FUNCTION_BLOCK I_Lighting (* Lighting Data LD *)
  (* Standard: ISO 11783-7; Classification: PGN 65088; Function: Lighting Data LD; Description: Copyright (c) 2024 HR Agrartechnik GmbH This program and the accompanying materials are made available under the terms of the Eclipse Public License 2.0 which is available at https://www.eclipse.org/legal/epl-2.0/ SPDX-License-Identifier: EPL-2.0 Message providing the status of all lighting functions of a tractor and connected implements. https://docs.ms-muc-docs.de/projects/isobus-other-docs/de/latest/PGN/PGN_65088.html *)
  (* Version 1.0, 2024-07-09, Franz Höpfinger, HR Agrartechnik GmbH *)
  PACKAGE isobus::tecu;
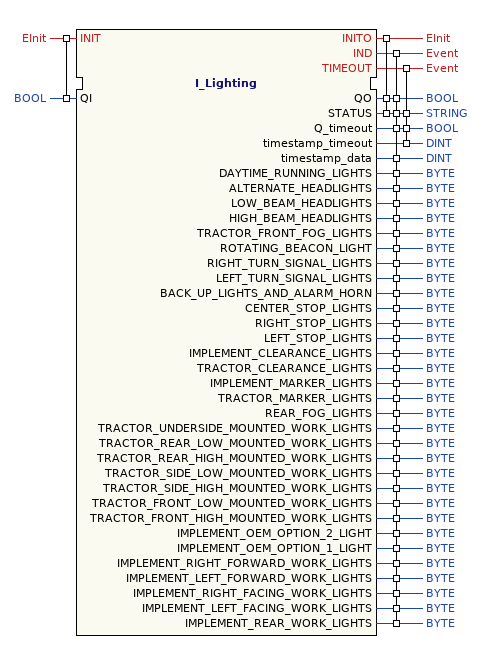
  EVENT_INPUT
    INIT : EInit WITH QI; (* Service Initialization *)
  END_EVENT
  EVENT_OUTPUT
    INITO : EInit WITH QO, STATUS; (* Initialization Confirm *)
    IND WITH QO, timestamp_data, STATUS, Q_timeout, DAYTIME_RUNNING_LIGHTS, ALTERNATE_HEADLIGHTS, LOW_BEAM_HEADLIGHTS, HIGH_BEAM_HEADLIGHTS, TRACTOR_FRONT_FOG_LIGHTS, ROTATING_BEACON_LIGHT, RIGHT_TURN_SIGNAL_LIGHTS, LEFT_TURN_SIGNAL_LIGHTS, BACK_UP_LIGHTS_AND_ALARM_HORN, CENTER_STOP_LIGHTS, RIGHT_STOP_LIGHTS, LEFT_STOP_LIGHTS, IMPLEMENT_CLEARANCE_LIGHTS, TRACTOR_CLEARANCE_LIGHTS, IMPLEMENT_MARKER_LIGHTS, TRACTOR_MARKER_LIGHTS, REAR_FOG_LIGHTS, TRACTOR_UNDERSIDE_MOUNTED_WORK_LIGHTS, TRACTOR_REAR_LOW_MOUNTED_WORK_LIGHTS, TRACTOR_REAR_HIGH_MOUNTED_WORK_LIGHTS, TRACTOR_SIDE_LOW_MOUNTED_WORK_LIGHTS, TRACTOR_SIDE_HIGH_MOUNTED_WORK_LIGHTS, TRACTOR_FRONT_LOW_MOUNTED_WORK_LIGHTS, TRACTOR_FRONT_HIGH_MOUNTED_WORK_LIGHTS, IMPLEMENT_OEM_OPTION_2_LIGHT, IMPLEMENT_OEM_OPTION_1_LIGHT, IMPLEMENT_RIGHT_FORWARD_WORK_LIGHTS, IMPLEMENT_LEFT_FORWARD_WORK_LIGHTS, IMPLEMENT_RIGHT_FACING_WORK_LIGHTS, IMPLEMENT_LEFT_FACING_WORK_LIGHTS, IMPLEMENT_REAR_WORK_LIGHTS; (* Indication from Resource *)
    TIMEOUT WITH timestamp_timeout, STATUS, Q_timeout;
  END_EVENT
  VAR_INPUT
    QI : BOOL; (* Event Input Qualifier *)
  END_VAR
  VAR_OUTPUT
    QO : BOOL; (* Event Output Qualifier *)
    STATUS : STRING;
    Q_timeout : BOOL;
    timestamp_timeout : DINT;
    timestamp_data : DINT;
    DAYTIME_RUNNING_LIGHTS : BYTE := BYTE#16#FF; (* Daytime running lights 2-bit QUARTER value (see Attributes for Details) *) {SET_ATTRIBUTE(SPN, 2404)} {SET_ATTRIBUTE(SP_Name, 'Daytime running lights')} {SET_ATTRIBUTE(SP_Position_In_PG, '1.1')} {SET_ATTRIBUTE(SP_Length, 2)} (* 2 bits *) {SET_ATTRIBUTE(Scaling, '4 states/2 bit')} {SET_ATTRIBUTE(Offset, )} {SET_ATTRIBUTE(Link, 'https://docs.ms-muc-docs.de/projects/isobus-other-docs/de/latest/PGN/PGN_65088.html#spn-2404-daytime-running-lights')}
    ALTERNATE_HEADLIGHTS : BYTE := BYTE#16#FF; (* Alternate headlights 2-bit QUARTER value (see Attributes for Details) *) {SET_ATTRIBUTE(SPN, 2352)} {SET_ATTRIBUTE(SP_Name, 'Alternate headlights')} {SET_ATTRIBUTE(SP_Position_In_PG, '1.3')} {SET_ATTRIBUTE(SP_Length, 2)} (* 2 bits *) {SET_ATTRIBUTE(Scaling, '4 states/2 bit')} {SET_ATTRIBUTE(Offset, )} {SET_ATTRIBUTE(Link, 'https://docs.ms-muc-docs.de/projects/isobus-other-docs/de/latest/PGN/PGN_65088.html#spn-2352-alternate-headlights')}
    LOW_BEAM_HEADLIGHTS : BYTE := BYTE#16#FF; (* Low-beam headlights 2-bit QUARTER value (see Attributes for Details) *) {SET_ATTRIBUTE(SPN, 2350)} {SET_ATTRIBUTE(SP_Name, 'Low-beam headlights')} {SET_ATTRIBUTE(SP_Position_In_PG, '1.5')} {SET_ATTRIBUTE(SP_Length, 2)} (* 2 bits *) {SET_ATTRIBUTE(Scaling, '4 states/2 bit')} {SET_ATTRIBUTE(Offset, )} {SET_ATTRIBUTE(Link, 'https://docs.ms-muc-docs.de/projects/isobus-other-docs/de/latest/PGN/PGN_65088.html#spn-2350-low-beam-headlights')}
    HIGH_BEAM_HEADLIGHTS : BYTE := BYTE#16#FF; (* High-beam headlights 2-bit QUARTER value (see Attributes for Details) *) {SET_ATTRIBUTE(SPN, 2348)} {SET_ATTRIBUTE(SP_Name, 'High-beam headlights')} {SET_ATTRIBUTE(SP_Position_In_PG, '1.7')} {SET_ATTRIBUTE(SP_Length, 2)} (* 2 bits *) {SET_ATTRIBUTE(Scaling, '4 states/2 bit')} {SET_ATTRIBUTE(Offset, )} {SET_ATTRIBUTE(Link, 'https://docs.ms-muc-docs.de/projects/isobus-other-docs/de/latest/PGN/PGN_65088.html#spn-2348-high-beam-headlights')}
    TRACTOR_FRONT_FOG_LIGHTS : BYTE := BYTE#16#FF; (* Tractor front fog lights 2-bit QUARTER value (see Attributes for Details) *) {SET_ATTRIBUTE(SPN, 2388)} {SET_ATTRIBUTE(SP_Name, 'Tractor front fog lights')} {SET_ATTRIBUTE(SP_Position_In_PG, '2.1')} {SET_ATTRIBUTE(SP_Length, 2)} (* 2 bits *) {SET_ATTRIBUTE(Scaling, '4 states/2 bit')} {SET_ATTRIBUTE(Offset, )} {SET_ATTRIBUTE(Link, 'https://docs.ms-muc-docs.de/projects/isobus-other-docs/de/latest/PGN/PGN_65088.html#spn-2388-tractor-front-fog-lights')}
    ROTATING_BEACON_LIGHT : BYTE := BYTE#16#FF; (* Rotating beacon light 2-bit QUARTER value (see Attributes for Details) *) {SET_ATTRIBUTE(SPN, 2386)} {SET_ATTRIBUTE(SP_Name, 'Rotating beacon light')} {SET_ATTRIBUTE(SP_Position_In_PG, '2.3')} {SET_ATTRIBUTE(SP_Length, 2)} (* 2 bits *) {SET_ATTRIBUTE(Scaling, '4 states/2 bit')} {SET_ATTRIBUTE(Offset, )} {SET_ATTRIBUTE(Link, 'https://docs.ms-muc-docs.de/projects/isobus-other-docs/de/latest/PGN/PGN_65088.html#spn-2386-rotating-beacon-light')}
    RIGHT_TURN_SIGNAL_LIGHTS : BYTE := BYTE#16#FF; (* Right-turn signal lights 2-bit QUARTER value (see Attributes for Details) *) {SET_ATTRIBUTE(SPN, 2370)} {SET_ATTRIBUTE(SP_Name, 'Right-turn signal lights')} {SET_ATTRIBUTE(SP_Position_In_PG, '2.5')} {SET_ATTRIBUTE(SP_Length, 2)} (* 2 bits *) {SET_ATTRIBUTE(Scaling, '4 states/2 bit')} {SET_ATTRIBUTE(Offset, )} {SET_ATTRIBUTE(Link, 'https://docs.ms-muc-docs.de/projects/isobus-other-docs/de/latest/PGN/PGN_65088.html#spn-2370-right-turn-signal-lights')}
    LEFT_TURN_SIGNAL_LIGHTS : BYTE := BYTE#16#FF; (* Left-turn signal lights 2-bit QUARTER value (see Attributes for Details) *) {SET_ATTRIBUTE(SPN, 2368)} {SET_ATTRIBUTE(SP_Name, 'Left-turn signal lights')} {SET_ATTRIBUTE(SP_Position_In_PG, '2.7')} {SET_ATTRIBUTE(SP_Length, 2)} (* 2 bits *) {SET_ATTRIBUTE(Scaling, '4 states/2 bit')} {SET_ATTRIBUTE(Offset, )} {SET_ATTRIBUTE(Link, 'https://docs.ms-muc-docs.de/projects/isobus-other-docs/de/latest/PGN/PGN_65088.html#spn-2368-left-turn-signal-lights')}
    BACK_UP_LIGHTS_AND_ALARM_HORN : BYTE := BYTE#16#FF; (* Back-up lights and alarm horn 2-bit QUARTER value (see Attributes for Details) *) {SET_ATTRIBUTE(SPN, 2392)} {SET_ATTRIBUTE(SP_Name, 'Back-up lights and alarm horn')} {SET_ATTRIBUTE(SP_Position_In_PG, '3.1')} {SET_ATTRIBUTE(SP_Length, 2)} (* 2 bits *) {SET_ATTRIBUTE(Scaling, '4 states/2 bit')} {SET_ATTRIBUTE(Offset, )} {SET_ATTRIBUTE(Link, 'https://docs.ms-muc-docs.de/projects/isobus-other-docs/de/latest/PGN/PGN_65088.html#spn-2392-back-up-lights-and-alarm-horn')}
    CENTER_STOP_LIGHTS : BYTE := BYTE#16#FF; (* Center stop lights 2-bit QUARTER value (see Attributes for Details) *) {SET_ATTRIBUTE(SPN, 2376)} {SET_ATTRIBUTE(SP_Name, 'Center stop lights')} {SET_ATTRIBUTE(SP_Position_In_PG, '3.3')} {SET_ATTRIBUTE(SP_Length, 2)} (* 2 bits *) {SET_ATTRIBUTE(Scaling, '4 states/2 bit')} {SET_ATTRIBUTE(Offset, )} {SET_ATTRIBUTE(Link, 'https://docs.ms-muc-docs.de/projects/isobus-other-docs/de/latest/PGN/PGN_65088.html#spn-2376-center-stop-lights')}
    RIGHT_STOP_LIGHTS : BYTE := BYTE#16#FF; (* Right stop lights 2-bit QUARTER value (see Attributes for Details) *) {SET_ATTRIBUTE(SPN, 2374)} {SET_ATTRIBUTE(SP_Name, 'Right stop lights')} {SET_ATTRIBUTE(SP_Position_In_PG, '3.5')} {SET_ATTRIBUTE(SP_Length, 2)} (* 2 bits *) {SET_ATTRIBUTE(Scaling, '4 states/2 bit')} {SET_ATTRIBUTE(Offset, )} {SET_ATTRIBUTE(Link, 'https://docs.ms-muc-docs.de/projects/isobus-other-docs/de/latest/PGN/PGN_65088.html#spn-2374-right-stop-lights')}
    LEFT_STOP_LIGHTS : BYTE := BYTE#16#FF; (* Left stop lights 2-bit QUARTER value (see Attributes for Details) *) {SET_ATTRIBUTE(SPN, 2372)} {SET_ATTRIBUTE(SP_Name, 'Left stop lights')} {SET_ATTRIBUTE(SP_Position_In_PG, '3.7')} {SET_ATTRIBUTE(SP_Length, 2)} (* 2 bits *) {SET_ATTRIBUTE(Scaling, '4 states/2 bit')} {SET_ATTRIBUTE(Offset, )} {SET_ATTRIBUTE(Link, 'https://docs.ms-muc-docs.de/projects/isobus-other-docs/de/latest/PGN/PGN_65088.html#spn-2372-left-stop-lights')}
    IMPLEMENT_CLEARANCE_LIGHTS : BYTE := BYTE#16#FF; (* Implement clearance lights 2-bit QUARTER value (see Attributes for Details) *) {SET_ATTRIBUTE(SPN, 2384)} {SET_ATTRIBUTE(SP_Name, 'Implement clearance lights')} {SET_ATTRIBUTE(SP_Position_In_PG, '4.1')} {SET_ATTRIBUTE(SP_Length, 2)} (* 2 bits *) {SET_ATTRIBUTE(Scaling, '4 states/2 bit')} {SET_ATTRIBUTE(Offset, )} {SET_ATTRIBUTE(Link, 'https://docs.ms-muc-docs.de/projects/isobus-other-docs/de/latest/PGN/PGN_65088.html#spn-2384-implement-clearance-lights')}
    TRACTOR_CLEARANCE_LIGHTS : BYTE := BYTE#16#FF; (* Tractor clearance lights 2-bit QUARTER value (see Attributes for Details) *) {SET_ATTRIBUTE(SPN, 2382)} {SET_ATTRIBUTE(SP_Name, 'Tractor clearance lights')} {SET_ATTRIBUTE(SP_Position_In_PG, '4.3')} {SET_ATTRIBUTE(SP_Length, 2)} (* 2 bits *) {SET_ATTRIBUTE(Scaling, '4 states/2 bit')} {SET_ATTRIBUTE(Offset, )} {SET_ATTRIBUTE(Link, 'https://docs.ms-muc-docs.de/projects/isobus-other-docs/de/latest/PGN/PGN_65088.html#spn-2382-tractor-clearance-lights')}
    IMPLEMENT_MARKER_LIGHTS : BYTE := BYTE#16#FF; (* Implement marker (position) lights 2-bit QUARTER value (see Attributes for Details) *) {SET_ATTRIBUTE(SPN, 2380)} {SET_ATTRIBUTE(SP_Name, 'Implement marker (position) lights')} {SET_ATTRIBUTE(SP_Position_In_PG, '4.5')} {SET_ATTRIBUTE(SP_Length, 2)} (* 2 bits *) {SET_ATTRIBUTE(Scaling, '4 states/2 bit')} {SET_ATTRIBUTE(Offset, )} {SET_ATTRIBUTE(Link, 'https://docs.ms-muc-docs.de/projects/isobus-other-docs/de/latest/PGN/PGN_65088.html#spn-2380-implement-marker-position-lights')}
    TRACTOR_MARKER_LIGHTS : BYTE := BYTE#16#FF; (* Tractor marker (position) lights 2-bit QUARTER value (see Attributes for Details) *) {SET_ATTRIBUTE(SPN, 2378)} {SET_ATTRIBUTE(SP_Name, 'Tractor marker (position) lights')} {SET_ATTRIBUTE(SP_Position_In_PG, '4.7')} {SET_ATTRIBUTE(SP_Length, 2)} (* 2 bits *) {SET_ATTRIBUTE(Scaling, '4 states/2 bit')} {SET_ATTRIBUTE(Offset, )} {SET_ATTRIBUTE(Link, 'https://docs.ms-muc-docs.de/projects/isobus-other-docs/de/latest/PGN/PGN_65088.html#spn-2378-tractor-marker-position-lights')}
    REAR_FOG_LIGHTS : BYTE := BYTE#16#FF; (* Rear fog lights 2-bit QUARTER value (see Attributes for Details) *) {SET_ATTRIBUTE(SPN, 2390)} {SET_ATTRIBUTE(SP_Name, 'Rear fog lights')} {SET_ATTRIBUTE(SP_Position_In_PG, '5.1')} {SET_ATTRIBUTE(SP_Length, 2)} (* 2 bits *) {SET_ATTRIBUTE(Scaling, '4 states/2 bit')} {SET_ATTRIBUTE(Offset, )} {SET_ATTRIBUTE(Link, 'https://docs.ms-muc-docs.de/projects/isobus-other-docs/de/latest/PGN/PGN_65088.html#spn-2390-rear-fog-lights')}
    TRACTOR_UNDERSIDE_MOUNTED_WORK_LIGHTS : BYTE := BYTE#16#FF; (* Tractor underside-mounted work lights 2-bit QUARTER value (see Attributes for Details) *) {SET_ATTRIBUTE(SPN, 2358)} {SET_ATTRIBUTE(SP_Name, 'Tractor underside-mounted work lights')} {SET_ATTRIBUTE(SP_Position_In_PG, '5.3')} {SET_ATTRIBUTE(SP_Length, 2)} (* 2 bits *) {SET_ATTRIBUTE(Scaling, '4 states/2 bit')} {SET_ATTRIBUTE(Offset, )} {SET_ATTRIBUTE(Link, 'https://docs.ms-muc-docs.de/projects/isobus-other-docs/de/latest/PGN/PGN_65088.html#spn-2358-tractor-underside-mounted-work-lights')}
    TRACTOR_REAR_LOW_MOUNTED_WORK_LIGHTS : BYTE := BYTE#16#FF; (* Tractor rear low-mounted work lights 2-bit QUARTER value (see Attributes for Details) *) {SET_ATTRIBUTE(SPN, 2360)} {SET_ATTRIBUTE(SP_Name, 'Tractor rear low-mounted work lights')} {SET_ATTRIBUTE(SP_Position_In_PG, '5.5')} {SET_ATTRIBUTE(SP_Length, 2)} (* 2 bits *) {SET_ATTRIBUTE(Scaling, '4 states/2 bit')} {SET_ATTRIBUTE(Offset, )} {SET_ATTRIBUTE(Link, 'https://docs.ms-muc-docs.de/projects/isobus-other-docs/de/latest/PGN/PGN_65088.html#spn-2360-tractor-rear-low-mounted-work-lights')}
    TRACTOR_REAR_HIGH_MOUNTED_WORK_LIGHTS : BYTE := BYTE#16#FF; (* Tractor rear high-mounted work lights 2-bit QUARTER value (see Attributes for Details) *) {SET_ATTRIBUTE(SPN, 2362)} {SET_ATTRIBUTE(SP_Name, 'Tractor rear high-mounted work lights')} {SET_ATTRIBUTE(SP_Position_In_PG, '5.7')} {SET_ATTRIBUTE(SP_Length, 2)} (* 2 bits *) {SET_ATTRIBUTE(Scaling, '4 states/2 bit')} {SET_ATTRIBUTE(Offset, )} {SET_ATTRIBUTE(Link, 'https://docs.ms-muc-docs.de/projects/isobus-other-docs/de/latest/PGN/PGN_65088.html#spn-2362-tractor-rear-high-mounted-work-lights')}
    TRACTOR_SIDE_LOW_MOUNTED_WORK_LIGHTS : BYTE := BYTE#16#FF; (* Tractor side low-mounted work lights 2-bit QUARTER value (see Attributes for Details) *) {SET_ATTRIBUTE(SPN, 2364)} {SET_ATTRIBUTE(SP_Name, 'Tractor side low-mounted work lights')} {SET_ATTRIBUTE(SP_Position_In_PG, '6.1')} {SET_ATTRIBUTE(SP_Length, 2)} (* 2 bits *) {SET_ATTRIBUTE(Scaling, '4 states/2 bit')} {SET_ATTRIBUTE(Offset, )} {SET_ATTRIBUTE(Link, 'https://docs.ms-muc-docs.de/projects/isobus-other-docs/de/latest/PGN/PGN_65088.html#spn-2364-tractor-side-low-mounted-work-lights')}
    TRACTOR_SIDE_HIGH_MOUNTED_WORK_LIGHTS : BYTE := BYTE#16#FF; (* Tractor side high-mounted work lights 2-bit QUARTER value (see Attributes for Details) *) {SET_ATTRIBUTE(SPN, 2366)} {SET_ATTRIBUTE(SP_Name, 'Tractor side high-mounted work lights')} {SET_ATTRIBUTE(SP_Position_In_PG, '6.3')} {SET_ATTRIBUTE(SP_Length, 2)} (* 2 bits *) {SET_ATTRIBUTE(Scaling, '4 states/2 bit')} {SET_ATTRIBUTE(Offset, )} {SET_ATTRIBUTE(Link, 'https://docs.ms-muc-docs.de/projects/isobus-other-docs/de/latest/PGN/PGN_65088.html#spn-2366-tractor-side-high-mounted-work-lights')}
    TRACTOR_FRONT_LOW_MOUNTED_WORK_LIGHTS : BYTE := BYTE#16#FF; (* Tractor front low-mounted work lights 2-bit QUARTER value (see Attributes for Details) *) {SET_ATTRIBUTE(SPN, 2354)} {SET_ATTRIBUTE(SP_Name, 'Tractor front low-mounted work lights')} {SET_ATTRIBUTE(SP_Position_In_PG, '6.5')} {SET_ATTRIBUTE(SP_Length, 2)} (* 2 bits *) {SET_ATTRIBUTE(Scaling, '4 states/2 bit')} {SET_ATTRIBUTE(Offset, )} {SET_ATTRIBUTE(Link, 'https://docs.ms-muc-docs.de/projects/isobus-other-docs/de/latest/PGN/PGN_65088.html#spn-2354-tractor-front-low-mounted-work-lights')}
    TRACTOR_FRONT_HIGH_MOUNTED_WORK_LIGHTS : BYTE := BYTE#16#FF; (* Tractor front high-mounted work lights 2-bit QUARTER value (see Attributes for Details) *) {SET_ATTRIBUTE(SPN, 2356)} {SET_ATTRIBUTE(SP_Name, 'Tractor front high-mounted work lights')} {SET_ATTRIBUTE(SP_Position_In_PG, '6.7')} {SET_ATTRIBUTE(SP_Length, 2)} (* 2 bits *) {SET_ATTRIBUTE(Scaling, '4 states/2 bit')} {SET_ATTRIBUTE(Offset, )} {SET_ATTRIBUTE(Link, 'https://docs.ms-muc-docs.de/projects/isobus-other-docs/de/latest/PGN/PGN_65088.html#spn-2356-tractor-front-high-mounted-work-lights')}
    IMPLEMENT_OEM_OPTION_2_LIGHT : BYTE := BYTE#16#FF; (* Implement OEM option 2 light 2-bit QUARTER value (see Attributes for Details) *) {SET_ATTRIBUTE(SPN, 2398)} {SET_ATTRIBUTE(SP_Name, 'Implement OEM option 2 light')} {SET_ATTRIBUTE(SP_Position_In_PG, '7.1')} {SET_ATTRIBUTE(SP_Length, 2)} (* 2 bits *) {SET_ATTRIBUTE(Scaling, '4 states/2 bit')} {SET_ATTRIBUTE(Offset, )} {SET_ATTRIBUTE(Link, 'https://docs.ms-muc-docs.de/projects/isobus-other-docs/de/latest/PGN/PGN_65088.html#spn-2398-implement-oem-option-2-light')}
    IMPLEMENT_OEM_OPTION_1_LIGHT : BYTE := BYTE#16#FF; (* Implement OEM option 1 light 2-bit QUARTER value (see Attributes for Details) *) {SET_ATTRIBUTE(SPN, 2396)} {SET_ATTRIBUTE(SP_Name, 'Implement OEM option 1 light')} {SET_ATTRIBUTE(SP_Position_In_PG, '7.3')} {SET_ATTRIBUTE(SP_Length, 2)} (* 2 bits *) {SET_ATTRIBUTE(Scaling, '4 states/2 bit')} {SET_ATTRIBUTE(Offset, )} {SET_ATTRIBUTE(Link, 'https://docs.ms-muc-docs.de/projects/isobus-other-docs/de/latest/PGN/PGN_65088.html#spn-2396-implement-oem-option-1-light')}
    IMPLEMENT_RIGHT_FORWARD_WORK_LIGHTS : BYTE := BYTE#16#FF; (* Implement right forward work lights 2-bit QUARTER value (see Attributes for Details) *) {SET_ATTRIBUTE(SPN, 2407)} {SET_ATTRIBUTE(SP_Name, 'Implement right forward work lights')} {SET_ATTRIBUTE(SP_Position_In_PG, '7.5')} {SET_ATTRIBUTE(SP_Length, 2)} (* 2 bits *) {SET_ATTRIBUTE(Scaling, '4 states/2 bit')} {SET_ATTRIBUTE(Offset, )} {SET_ATTRIBUTE(Link, 'https://docs.ms-muc-docs.de/projects/isobus-other-docs/de/latest/PGN/PGN_65088.html#spn-2407-implement-right-forward-work-lights')}
    IMPLEMENT_LEFT_FORWARD_WORK_LIGHTS : BYTE := BYTE#16#FF; (* Implement left forward work lights 2-bit QUARTER value (see Attributes for Details) *) {SET_ATTRIBUTE(SPN, 2598)} {SET_ATTRIBUTE(SP_Name, 'Implement left forward work lights')} {SET_ATTRIBUTE(SP_Position_In_PG, '7.7')} {SET_ATTRIBUTE(SP_Length, 2)} (* 2 bits *) {SET_ATTRIBUTE(Scaling, '4 states/2 bit')} {SET_ATTRIBUTE(Offset, )} {SET_ATTRIBUTE(Link, 'https://docs.ms-muc-docs.de/projects/isobus-other-docs/de/latest/PGN/PGN_65088.html#spn-2598-implement-left-forward-work-lights')}
    IMPLEMENT_RIGHT_FACING_WORK_LIGHTS : BYTE := BYTE#16#FF; (* Implement right-facing work lights 2-bit QUARTER value (see Attributes for Details) *) {SET_ATTRIBUTE(SPN, 2402)} {SET_ATTRIBUTE(SP_Name, 'Implement right-facing work lights')} {SET_ATTRIBUTE(SP_Position_In_PG, '8.3')} {SET_ATTRIBUTE(SP_Length, 2)} (* 2 bits *) {SET_ATTRIBUTE(Scaling, '4 states/2 bit')} {SET_ATTRIBUTE(Offset, )} {SET_ATTRIBUTE(Link, 'https://docs.ms-muc-docs.de/projects/isobus-other-docs/de/latest/PGN/PGN_65088.html#spn-2402-implement-right-facing-work-lights')}
    IMPLEMENT_LEFT_FACING_WORK_LIGHTS : BYTE := BYTE#16#FF; (* Implement left-facing work lights 2-bit QUARTER value (see Attributes for Details) *) {SET_ATTRIBUTE(SPN, 2400)} {SET_ATTRIBUTE(SP_Name, 'Implement left-facing work lights')} {SET_ATTRIBUTE(SP_Position_In_PG, '8.5')} {SET_ATTRIBUTE(SP_Length, 2)} (* 2 bits *) {SET_ATTRIBUTE(Scaling, '4 states/2 bit')} {SET_ATTRIBUTE(Offset, )} {SET_ATTRIBUTE(Link, 'https://docs.ms-muc-docs.de/projects/isobus-other-docs/de/latest/PGN/PGN_65088.html#spn-2400-implement-left-facing-work-lights')}
    IMPLEMENT_REAR_WORK_LIGHTS : BYTE := BYTE#16#FF; (* Implement rear work lights 2-bit QUARTER value (see Attributes for Details) *) {SET_ATTRIBUTE(SPN, 2394)} {SET_ATTRIBUTE(SP_Name, 'Implement rear work lights')} {SET_ATTRIBUTE(SP_Position_In_PG, '8.7')} {SET_ATTRIBUTE(SP_Length, 2)} (* 2 bits *) {SET_ATTRIBUTE(Scaling, '4 states/2 bit')} {SET_ATTRIBUTE(Offset, )} {SET_ATTRIBUTE(Link, 'https://docs.ms-muc-docs.de/projects/isobus-other-docs/de/latest/PGN/PGN_65088.html#spn-2394-implement-rear-work-lights')}
  END_VAR
END_FUNCTION_BLOCK
